// Mitsubishi GX Works2 project: Modbus TCP 통합   PLC: Q03UDV

PROGRAM MAIN
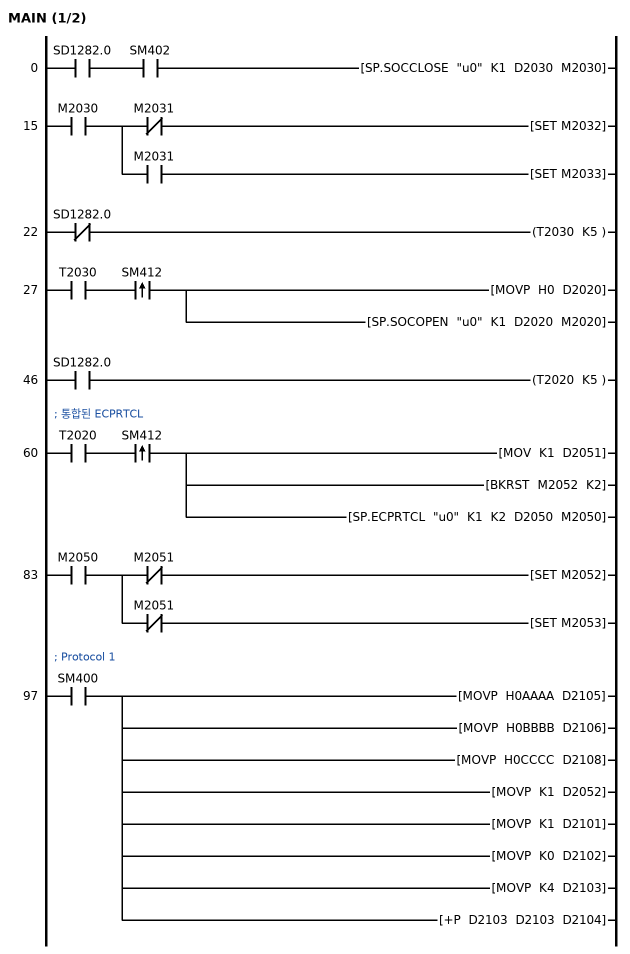
0     LD      SD1282.0
      AND     SM402
      SP.SOCCLOSE "u0" K1 D2030 M2030
15    LD      M2030
      MPS
      ANI     M2031
      SET     M2032
      MPP
      AND     M2031
      SET     M2033
22    LDI     SD1282.0
      OUT     T2030 K5
27    LD      T2030
      ANDP    SM412
      MOVP    H0 D2020
      SP.SOCOPEN "u0" K1 D2020 M2020
46    LD      SD1282.0
      OUT     T2020 K5
; 통합된 ECPRTCL
60    LD      T2020
      ANDP    SM412
      MOV     K1 D2051
      BKRST   M2052 K2
      SP.ECPRTCL "u0" K1 K2 D2050 M2050
83    LD      M2050
      MPS
      ANI     M2051
      SET     M2052
      MPP
      ANI     M2051
      SET     M2053
; Protocol 1
97    LD      SM400
      MOVP    H0AAAA D2105
      MOVP    H0BBBB D2106
      MOVP    H0CCCC D2108
      MOVP    K1 D2052
      MOVP    K1 D2101
      MOVP    K0 D2102
      MOVP    K4 D2103
      +P      D2103 D2103 D2104
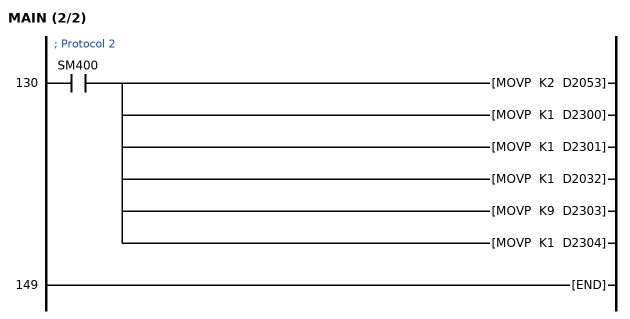
; Protocol 2
130   LD      SM400
      MOVP    K2 D2053
      MOVP    K1 D2300
      MOVP    K1 D2301
      MOVP    K1 D2032
      MOVP    K9 D2303
      MOVP    K1 D2304
149   END
END_PROGRAM
